# EPICS autosave request: support/dxp-s55/dxpApp/Db/dxpMED_settings.req
$(P)PresetMode
$(P)PresetReal
$(P)PresetLive
$(P)PresetEvents
$(P)PresetTriggers
$(P)StatusAll.SCAN
$(P)ReadAll.SCAN
$(P)TraceTimes
$(P)TraceModes
$(P)EnableClientWait
